// TIA Portal V17 export
// export: Created 2025-06-26T07:49:16.2345184Z, ExportSetting WithDefaults, DisplayName Totally Integrated Automation Portal, DisplayVersion V17 Update 8, DisplayName TIA Portal Openness, DisplayVersion V17 Update 8, DisplayName TIA Portal Version Control Interface, DisplayVersion V17, DisplayName STEP 7 Professional, DisplayVersion V17 Update 8, DisplayName STEP 7 Safety, DisplayVersion V17 Update 6, DisplayName WinCC Advanced, DisplayVersion V17 Update 8
FUNCTION_BLOCK "InputProcessing"   // FB48, FBD
{ S7_Optimized_Access := 'TRUE' }
AUTHOR : Heaten
VERSION : 0.1
// stored: AutoNumber false, IsIECCheckEnabled false, IsRetainMemResEnabled false, MemoryReserve 0, SetENOAutomatically false, UDAEnableTagReadback false
   VAR
      PumaInputProcessing : "PumaInputProcessing";
      CustomerInputProcessing { S7_SetPoint := 'True'} : "CustomerInputProcessing";
   END_VAR
BEGIN

REGION Network 1: Values from Puma
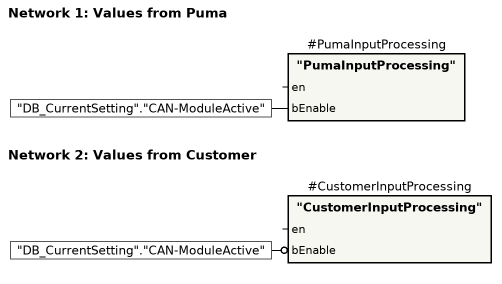
   #PumaInputProcessing(bEnable := "DB_CurrentSetting"."CAN-ModuleActive");   // "PumaInputProcessing"
END_REGION

REGION Network 2: Values from Customer
   #CustomerInputProcessing(bEnable := NOT "DB_CurrentSetting"."CAN-ModuleActive");   // "CustomerInputProcessing"
END_REGION

REGION Network 3: Analog inputs
   // Directly connected
END_REGION

REGION Network 4: Digital inputs
   // Directly connected
END_REGION
END_FUNCTION_BLOCK
